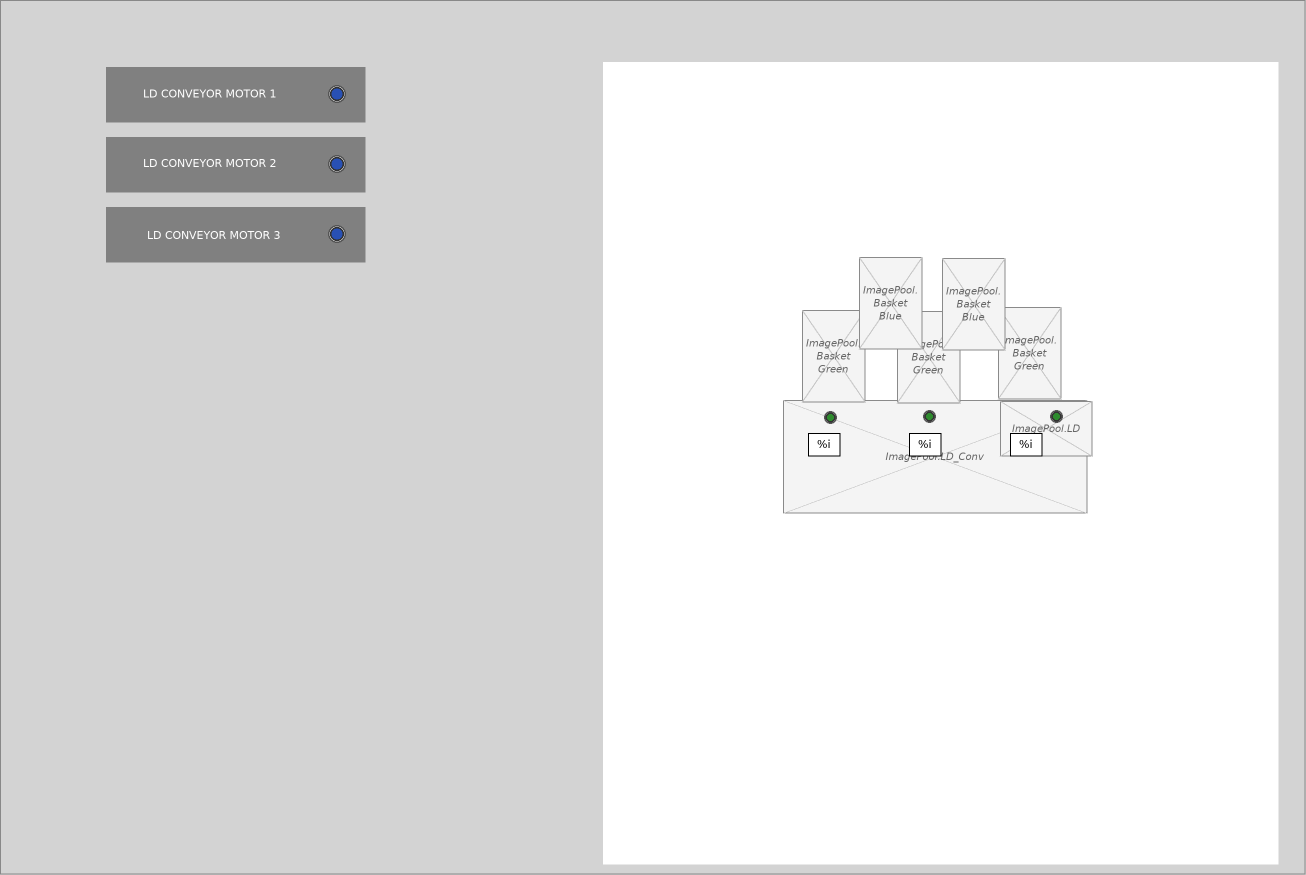
VISUALIZATION Auto_Loading  // 1306x875
    Rectangle (0,0 1306x875)
    Rectangle (603,62 675x802)
    RoundedRectangle (106,67 259x55)
    Label (140,69 176x50), "LD CONVEYOR MOTOR 1"
    Lamp1 (327,84 20x20), variable: ARdsMAP_HmiVariableGeneral.bLdConveyorMotor01_IND, style: Lamp-Lamp1-Blue
    RoundedRectangle (106,137 259x55)
    Label (140,136 178x55), "LD CONVEYOR MOTOR 2"
    Lamp1 (327,154 20x20), variable: ARdsMAP_HmiVariableGeneral.bLdConveyorMotor02_IND, style: Lamp-Lamp1-Blue
    RoundedRectangle (106,207 259x55)
    Label (144,208 176x55), "LD CONVEYOR MOTOR 3"
    Lamp1 (327,224 20x20), variable: ARdsMAP_HmiVariableGeneral.bLdConveyorMotor03_IND, style: Lamp-Lamp1-Blue
    Image (783,400 304x113), image: ImagePool.LD_Conv
    Image (998,307 63x92), invisible if: NOT.ARbBasketGdFlag[1], image: ImagePool.Basket Green
        OnMouseDown: execute { AR2sDSCv_LdConfirmBasketInfo[1,3].iProductRecipeNo:=0; }
    Image (802,310 63x92), invisible if: NOT AR2sDSCv_LdConfirmBasketInfo[1,1].bAvailibility, image: ImagePool.Basket Green
        OnMouseDown: execute { AR2sDSCv_LdConfirmBasketInfo[1,1].iProductRecipeNo:=0; }
    Image (1000,401 92x55), image: ImagePool.LD
    Image (897,311 63x92), invisible if: NOT AR2sDSCv_LdConfirmBasketInfo[1,2].bAvailibility, image: ImagePool.Basket Green
        OnMouseDown: execute { AR2sDSCv_LdConfirmBasketInfo[1,2].iProductRecipeNo:=0; }
    Image (859,257 63x92), invisible if: NOT AR2sDSCv_LdTransferBasketInfo[1,1].bAvailibility, image: ImagePool.Basket Blue
        OnMouseDown: execute { AR2sDSCv_LdTransferBasketInfo[1,1].iProductRecipeNo:=0; }
    Image (942,258 63x92), invisible if: NOT AR2sDSCv_LdTransferBasketInfo[1,2].bAvailibility, image: ImagePool.Basket Blue
        OnMouseDown: execute { AR2sDSCv_LdTransferBasketInfo[1,2].iProductRecipeNo:=0;; }
    Lamp1 (823,410 15x15), variable: ARdsMAP_HmiVariableGeneral.bLdFeedSensor_IND, style: Lamp-Lamp1-Green
    Lamp1 (1049,409 15x15), variable: ARdsMAP_HmiVariableGeneral.bLdPickSensor_IND, style: Lamp-Lamp1-Green
    Lamp1 (922,409 15x15), variable: ARdsMAP_HmiVariableGeneral.bLdIndex1Sensor_IND, style: Lamp-Lamp1-Green
    Rectangle (909,433 32x23), "%i", text variable: AR2sDSCv_LdConfirmBasketInfo[1,2].iProductRecipeNo
        OnMouseDown: write the text variable via VisuDialogs.Numpad
    Rectangle (1010,433 32x23), "%i", text variable: AR2sDSCv_LdConfirmBasketInfo[1,3].iProductRecipeNo
        OnMouseDown: write the text variable via VisuDialogs.Numpad
    Rectangle (808,433 32x23), "%i", text variable: AR2sDSCv_LdConfirmBasketInfo[1,1].iProductRecipeNo
        OnMouseDown: write the text variable via VisuDialogs.Numpad
END_VISUALIZATION

(* stored: Version 1.1.0.1, ProductVersion 3.1.4024.12
   Visu Auto_Loading: Id {dcffa3e2-a065-4e6c-8122-5aa603743c82} *)
